PROGRAM MAIN
VAR
END_VAR

END_PROGRAM

(* stored: Version 1.1.0.1, ProductVersion 3.1.4024.13
   POU MAIN: Id {9162ce8e-240e-4f99-abe8-990f4b0301ee}, SpecialFunc None *)
